PROGRAM P_Section_1
VAR
END_VAR

P_Example_1_TONs();
P_Example_2_TOFs();
P_Example_3_TPs();

END_PROGRAM

(* stored: Version 1.1.0.1, ProductVersion 3.1.4024.4
   POU P_Section_1: Id {6b528a2e-6c61-400c-b708-26ec986ea447}, SpecialFunc None *)
